PROGRAM ElevationControl
VAR_INPUT
	up:	BOOL;
	down: BOOL;
	reset: BOOL;
	enable :  BOOL;
END_VAR

VAR
	ElevationAxisJog:	FB_AxisJog;
	ElevationAxis:		FB_Axis;
	error: BOOL;
	position: LREAL;
	act_position: LREAL;
END_VAR

IF PendantControl.manual THEN
	ElevationAxisJog(	bPowerEnable := enable AND Main.power_OK,
						bEnable_Positive := GVL_Telescope.brake_azimuth_eve,
						bEnable_Negative := GVL_Telescope.brake_azimuth_eve,
						bForward := up,
						bBackward := down,
						bReset := reset,
						bStop := up AND down,
						bErr => error,
						fActPos => act_position,
						stAxis :=	GVL_Telescope.ElevationAxisRef);	
ELSE
	ElevationAxis(	bPowerEnable := TelescopeControl.power AND Main.power_OK,
					bReset := reset,
					fMoveAbsPos := position, 
					fActPos => act_position,
					bAxError => error,
					stAxis :=	GVL_Telescope.ElevationAxisRef);
END_IF

END_PROGRAM

(* stored: Version 1.1.0.1, ProductVersion 3.1.4024.0
   POU ElevationControl: Id {c0371b19-3d1d-4f20-bd19-ce60539d69cd}, SpecialFunc None *)
